# EPICS substitutions: db/Beckhoff_3XXX/ecmcEL3702_s100.substitutions
file "ecmcEcSlave.template"
{
  pattern {}
          {}
}

file "ecmcEL37XX-chX.template"
{
  pattern {CH_ID, DTYP,             FTVL,  NELM }
          {1,     asynInt16ArrayIn, SHORT, 100  }
          {2,     asynInt16ArrayIn, SHORT, 100  }
}
